// TIA Portal project "Simulation1.1" (V15)

(* hardware
DEVICE "S7-1200 station_1"  S7-1200 Station
   slot 0: "Rack_0"  S7-1200 Rack  Rack  V1.0
   slot 1: "PLC_1"  CPU 1214C DC/DC/DC  6ES7 214-1AG40-0XB0  V4.2
*)

// ===== PLC "PLC_1"  CPU 1214C DC/DC/DC =====

VAR_GLOBAL   // PLC tag table "Default tag table"
   ""Takeoff_at_End3"" AT %I0.5 : Bool;
   ""Regulation"" AT %I0.6 : Bool;
   ""Conveyor_Belt_1_Input"" AT %I0.1 : Bool;
   ""Conveyor_Belt_2_Input"" AT %I0.2 : Bool;
   ""Conveyor_Belt_3_Input"" AT %I0.3 : Bool;
   ""Conveyor_Belt_3_Confirm"" AT %I0.4 : Bool;
   ""Emergency_3_Confirm"" AT %I1.2 : Bool;
   ""Emergency_2_Confirm"" AT %I1.1 : Bool;
   ""Emergency_1_Confirm"" AT %I1.0 : Bool;
   ""Conveyor_Belt_1_Output"" AT %Q0.1 : Bool;
   ""Conveyor_Belt_2_Output"" AT %Q0.2 : Bool;
   ""Conveyor_Belt_3_Output"" AT %Q0.3 : Bool;
   ""Conveyor_Belt_2_Status"" AT %Q0.5 : Bool;
   ""Conveyor_Belt_3_Status"" AT %Q0.6 : Bool;
   ""Conveyor_Belt_1_Status"" AT %Q0.4 : Bool;
   ""Conveyor_Belt_1_Alarm"" AT %Q1.0 : Bool;
   ""Conveyor_Belt_2_Alarm"" AT %Q1.1 : Bool;
   ""Conveyor_Belt_3_Alarm"" AT %Q1.2 : Bool;
END_VAR